ABB RobotStudio station: Practica2_20220428-135920.rsstn

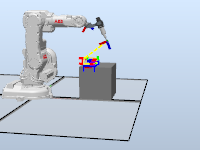
Station Practica2 (saved by RobotStudio 20.4.9280.0)
Controller Controlador3
  mechanical unit ROB_1: IRB140_6_81_C_03, 6 joints, base frame (0, 0, 0) mm
Layout (positions relative to the parent item):
  - IRB140_6_81_C_03 [mechanism, from Robots\IRB140_6_81_C_G_03.rslib] at (0, 0, 0) mm; joint values [-0.2106, -0.1182, 0.5465, 1.2645, 0.8026, -0.7606] (rad or m)
  - MyTool [mechanism, from Training Objects\myTool.rslib] at (506.28, -3.19, 679.5) mm, rotated rx 180 ry 60 rz 179.64 deg
  - Pieza_1 [part]
  - Pieza_6 [part]
Attachment: MyTool is attached to IRB140_6_81_C_03 / Link6
Attachment: Workobject_2 is attached to Pieza_6
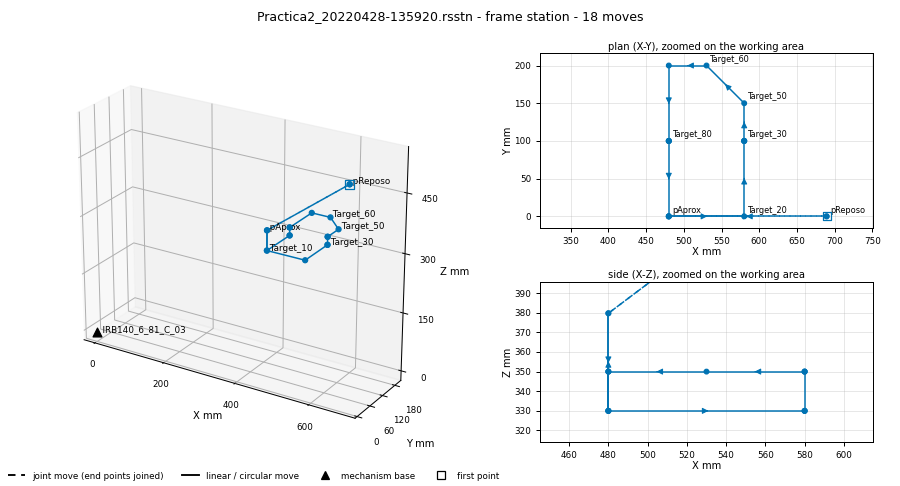
[picture p0: tool path of Practica2_20220428-135920.rsstn in frame station, 18 of 18 moves have a stored position in this frame; points joined in program order, loops and branches not executed]
Targets, tools, work objects and paths stored in the station, written as RAPID:
! task (no controller)
MODULE CalibData
  TASK PERS wobjdata Workobject_1:=[FALSE,TRUE,"",[[480,0,300],[1,0,0,0]],[[0,0,0],[1,0,0,0]]];
ENDMODULE

! task T_ROB1
MODULE CalibData
  PERS tooldata MyTool:=[TRUE,[[31.792631019,0,229.638935148],[0.945518576,0,0.325568154,0]],[1,[0,0,1],[1,0,0,0],0,0,0]];
  TASK PERS wobjdata Workobject_2:=[FALSE,TRUE,"",[[480,0,300],[1,0,0,0]],[[0,0,0],[1,0,0,0]]];
ENDMODULE

! task T_ROB1
MODULE Module1
  CONST robtarget Target_10:=[[0,0,30],[0,0,1,0],[0,0,-1,0],[9E+09,9E+09,9E+09,9E+09,9E+09,9E+09]];
  CONST robtarget Target_20:=[[100,0,30],[0,0,1,0],[0,0,-1,0],[9E+09,9E+09,9E+09,9E+09,9E+09,9E+09]];
  CONST robtarget Target_30:=[[100,100,30],[0,0,1,0],[0,-1,0,0],[9E+09,9E+09,9E+09,9E+09,9E+09,9E+09]];
  CONST robtarget Target_40:=[[100,100,50],[0,0,1,0],[0,-1,0,0],[9E+09,9E+09,9E+09,9E+09,9E+09,9E+09]];
  CONST robtarget Target_50:=[[100,150.001,50],[0,0,1,0],[0,-1,0,0],[9E+09,9E+09,9E+09,9E+09,9E+09,9E+09]];
  CONST robtarget Target_60:=[[50,200,50],[0,0,1,0],[0,-1,0,0],[9E+09,9E+09,9E+09,9E+09,9E+09,9E+09]];
  CONST robtarget Target_70:=[[0,200,50],[0,0,1,0],[0,-1,0,0],[9E+09,9E+09,9E+09,9E+09,9E+09,9E+09]];
  CONST robtarget Target_80:=[[0,100,50],[0,0,1,0],[0,-1,0,0],[9E+09,9E+09,9E+09,9E+09,9E+09,9E+09]];
  CONST robtarget Target_90:=[[0,100,30],[0,0,1,0],[0,-1,0,0],[9E+09,9E+09,9E+09,9E+09,9E+09,9E+09]];
  CONST robtarget pAprox:=[[0.000010305,0,79.717534108],[-0.000000111,0,1,0],[0,0,-1,0],[9E+09,9E+09,9E+09,9E+09,9E+09,9E+09]];
  CONST robtarget pReposo:=[[689.268487273,0,537.14730631],[0.190808996,0,0.981627183,0],[0,0,0,0],[9E+09,9E+09,9E+09,9E+09,9E+09,9E+09]];
  CONST robtarget Target_30_girar:=[[100,100,30],[0,0,0.923879533,0.382683432],[-1,0,-1,0],[9E+09,9E+09,9E+09,9E+09,9E+09,9E+09]];
  CONST robtarget Target_40_girar:=[[100,100,50],[0,0,0.923879533,0.382683432],[-1,0,-1,0],[9E+09,9E+09,9E+09,9E+09,9E+09,9E+09]];
  CONST robtarget Target_80_girar:=[[0,100,50],[0,0,0.923879533,0.382683432],[-1,0,-1,0],[9E+09,9E+09,9E+09,9E+09,9E+09,9E+09]];
  CONST robtarget Target_90_girar:=[[0,100,30],[0,0,0.923879533,0.382683432],[-1,0,-1,0],[9E+09,9E+09,9E+09,9E+09,9E+09,9E+09]];
  PROC Path_10()
    MoveJ pReposo,v1000,z100,MyTool\WObj:=wobj0;
    MoveJ pAprox,v1000,z100,MyTool\WObj:=Workobject_2;
    MoveL Target_10,v100,z0,MyTool\WObj:=Workobject_2;
    MoveL Target_20,v100,z0,MyTool\WObj:=Workobject_2;
    MoveL Target_30,v100,z0,MyTool\WObj:=Workobject_2;
    MoveL Target_30_girar,v100,z100,MyTool\WObj:=Workobject_2;
    MoveL Target_40_girar,v100,z100,MyTool\WObj:=Workobject_2;
    MoveL Target_40,v100,z0,MyTool\WObj:=Workobject_2;
    MoveL Target_50,v100,z0,MyTool\WObj:=Workobject_2;
    MoveL Target_60,v100,z0,MyTool\WObj:=Workobject_2;
    MoveL Target_70,v100,z0,MyTool\WObj:=Workobject_2;
    MoveL Target_80,v100,z0,MyTool\WObj:=Workobject_2;
    MoveL Target_80_girar,v100,z100,MyTool\WObj:=Workobject_2;
    MoveL Target_90_girar,v100,z100,MyTool\WObj:=Workobject_2;
    MoveL Target_90,v100,z0,MyTool\WObj:=Workobject_2;
    MoveL Target_10,v100,z0,MyTool\WObj:=Workobject_2;
    MoveL pAprox,v200,z100,MyTool\WObj:=Workobject_2;
    MoveJ pReposo,v1000,z100,MyTool\WObj:=wobj0;
  ENDPROC
ENDMODULE

